// Brief: Setup Arm Init
FUNCTION_BLOCK PUBLIC FB_SetupCtrlInit EXTENDS FB_SetupArmCtrlBase
VAR_INPUT
END_VAR
VAR_OUTPUT
END_VAR
VAR
	m_initState :INT :=0;
END_VAR

// override this function in each exact controller
METHOD PROTECTED calcCmdJntPos : BOOL
VAR_IN_OUT CONSTANT
	i_setupArm	:FB_SetupArm;
END_VAR


VAR 
	i :INT;
	curJntVel :Vec5d;
END_VAR
END_METHOD

METHOD PUBLIC init : BOOL
VAR_IN_OUT CONSTANT
	i_setupArm	:FB_SetupArm;
END_VAR
VAR_IN_OUT 
	r_setupArmCtrlCmd :ST_SetupArmCtrlCmds;
END_VAR


VAR
	i:INT;
END_VAR
SUPER^.Init(i_setupArm,r_setupArmCtrlCmd);
END_METHOD

END_FUNCTION_BLOCK

(* stored: Version 1.1.0.1, ProductVersion 3.1.4024.12
   POU FB_SetupCtrlInit: Id {eac05193-39e5-4249-a95b-72d2422e8330}, SpecialFunc None
   Method calcCmdJntPos: Id {1e0a883f-c826-468a-9931-3e424876db21}
   Method init: Id {dbcec065-8704-4c57-a097-e13d35679382} *)
